TYPE (* logiBUS_DI Struct *)
  (* Version 1.0, 2025-07-21, Franz Höpfinger, initial API and implementation and/or initial documentation *)
  PACKAGE logiBUS::io::DI;
  IMPORT eclipse4diac::core::TypeHash;
  logiBUS_DI_Events_S : STRUCT
    EType : USINT := 255;
  END_STRUCT;
END_TYPE
